TYPE csp_main_accuChange_RFID_running_check_status :
(
	READ_RUNNING_CHECK_STATUS_START									:= 0,
	READ_RUNNING_CHECK_STATUS_EOAT_CHECK_CP							:= 1,
	READ_RUNNING_CHECK_STATUS_EOAT_SEND_READ						:= 2,
	READ_RUNNING_CHECK_STATUS_EOAT_CHECK_READ						:= 3,
	READ_RUNNING_CHECK_STATUS_LOADER_PUSHER_CHECK_CP				:= 4,
	READ_RUNNING_CHECK_STATUS_LOADER_PUSHER_SEND_READ				:= 5,
	READ_RUNNING_CHECK_STATUS_LOADER_PUSHER_CHECK_READ				:= 6,
	READ_RUNNING_CHECK_STATUS_LOADER_PLATE_CHECK_CP					:= 7,
	READ_RUNNING_CHECK_STATUS_LOADER_PLATE_SEND_READ				:= 8,
	READ_RUNNING_CHECK_STATUS_LOADER_PLATE_CHECK_READ				:= 9,
	
	READ_RUNNING_CHECK_STATUS_DONE									:= 900,
	READ_RUNNING_CHECK_STATUS_WAITING								:= 950,
	READ_RUNNING_CHECK_STATUS_ERROR									:= 999
):= READ_RUNNING_CHECK_STATUS_WAITING;
END_TYPE

(* stored: Version 1.1.0.1, ProductVersion 3.1.4024.3
   DUT csp_main_accuChange_RFID_running_check_status: Id {680ed942-29ad-0062-3fd5-9f1d6cdb73b3} *)
